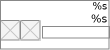
VISUALIZATION VIS_SENSOR_ROUND_RightAboveCheckQuerry  // 110x50
VAR_INPUT
    ITF_SENSOR_IN   :   ITF_SENSOR;
	stExklParameter	:	STRING [40];	
END_VAR
    Frame (0,0 110x50)
        shows VIS_SENSOR_ROUND_RightAboveCheckIsEnabled(ITF_SENSOR_IN := ITF_SENSOR_IN, stExklParameter := stExklParameter)
END_VISUALIZATION

// 40 Visualizations/ICON/SENSOR_FLAT/SENSOR_FLAT_TXT_RIGHT/BELOW/VIS_SENSOR_FLAT_RIGHT_BELOW
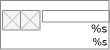
VISUALIZATION VIS_SENSOR_FLAT_RIGHT_BELOW  // 110x50
VAR_INPUT
    ITF_SENSOR_IN   :   ITF_SENSOR;	
END_VAR
VAR_INPUT CONSTANT	
	stExklParameter	:	STRING [40] := ' ';	
END_VAR
VAR CONSTANT
	uiIconNr		:	UINT := 3;
END_VAR
    Frame (0,0 110x50), invisible if: NOT fcCheckQuerryAndIconReturn(_ITF_IN := ITF_SENSOR_IN, _uiIconNr_IN := uiIconNr)
        shows VIS_SENSOR_FLAT_RigthBelowCheckQuerry(ITF_SENSOR_IN := ITF_SENSOR_IN, stExklParameter := stExklParameter)
END_VISUALIZATION

// 40 Visualizations/ICON/SENSOR_FLAT/SENSOR_FLAT_TXT_RIGHT/BELOW/VIS_SENSOR_FLAT_RigthBelowCheckIsEnabled
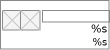
VISUALIZATION VIS_SENSOR_FLAT_RigthBelowCheckIsEnabled  // 110x50
VAR_INPUT
    ITF_SENSOR_IN   :   ITF_SENSOR;
	stExklParameter	:	STRING [40];	
END_VAR
    Frame (2,10 38x20), invisible if: NOT ITF_SENSOR_IN.proIsEnabled
        shows SensorFlat(ITF_SENSORIN := ITF_SENSOR_IN)
    Frame (42,10 68x40), invisible if: NOT ITF_SENSOR_IN.proIsEnabled
        shows ValueDwnUp(ITF_SENSORIN := ITF_SENSOR_IN, uiTextAusrichtung := 4)
    Rectangle (0,0 110x50)
        OnMouseClick:  Dialog=POPUP_SENSOR, Parameters={stExklParameter: stExklParameter, ITF_SENSORIN: ITF_SENSOR_IN, uiPopUpGruppe: 0}, OpenCentered=True
END_VISUALIZATION

// 40 Visualizations/ICON/SENSOR_FLAT/SENSOR_FLAT_TXT_RIGHT/BELOW/VIS_SENSOR_FLAT_RigthBelowCheckQuerry
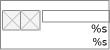
VISUALIZATION VIS_SENSOR_FLAT_RigthBelowCheckQuerry  // 110x50
VAR_INPUT
    ITF_SENSOR_IN   :   ITF_SENSOR;	
	stExklParameter	:	STRING [40];	
END_VAR
    Frame (0,0 110x50)
        shows VIS_SENSOR_FLAT_RigthBelowCheckIsEnabled(ITF_SENSOR_IN := ITF_SENSOR_IN, stExklParameter := stExklParameter)
END_VISUALIZATION

// 40 Visualizations/ICON/SENSOR_ROUND/SENSOR_ROUND_TXT_RIGHT/BELOW/VIS_SENSOR_ROUND_RIGHT_BELOW
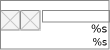
VISUALIZATION VIS_SENSOR_ROUND_RIGHT_BELOW  // 110x50
VAR_INPUT
    ITF_SENSOR_IN   :   ITF_SENSOR;	
END_VAR
VAR_INPUT CONSTANT	
	stExklParameter	:	STRING [40] := ' ';	
END_VAR
VAR CONSTANT
	uiIconNr		:	UINT := 5;
END_VAR
    Frame (0,0 110x50), invisible if: NOT fcCheckQuerryAndIconReturn(_ITF_IN := ITF_SENSOR_IN, _uiIconNr_IN := uiIconNr)
        shows VIS_SENSOR_ROUND_RightBelowCheckQuerry(ITF_SENSOR_IN := ITF_SENSOR_IN, stExklParameter := stExklParameter)
END_VISUALIZATION

// 40 Visualizations/ICON/SENSOR_BASE/ICON/Value/ValueDwnUp
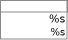
VISUALIZATION ValueDwnUp  // 68x40
VAR_INPUT
    ITF_SENSORIN   :   ITF_SENSOR;	
END_VAR
VAR_INPUT CONSTANT
    uiTextAusrichtung   : UINT := 4;    // 0 = Oben links | 1 = Horizontal zentriert | 2 = Rechts | 4 = Vertikal zentriert | 8 = Unten
END_VAR
    Frame (0,0 68x12)
        shows CtaSysSensorReCalculation.ValueRC(ITF_SENSOR_RE_CALCULATE := ITF_SENSORIN.ITF_RC, uiTextAusrichtung := uiTextAusrichtung)
    Textfield (0,13 68x12), "%s", text variable: ITF_SENSORIN.proSoftwareValue
        p3718999670: uiTextAusrichtung
    Textfield (0,26 68x12), "%s", text variable: ITF_SENSORIN.proGetBMK, invisible if: ITF_SENSORIN.proNoBmkInList
        p3718999670: uiTextAusrichtung
END_VISUALIZATION

// 40 Visualizations/ICON/SENSOR_BASE/ICON/Round/SensorRound
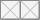
VISUALIZATION SensorRound  // 40x20
VAR_INPUT
    ITF_SENSORIN   :   ITF_SENSOR;	
END_VAR
    Ellipse (10,0 20x20), colour toggle: ITF_SENSORIN.proAcknowlege, invisible if: ITF_SENSORIN.proIsError
    Ellipse (10,0 20x20), colour toggle: ITF_SENSORIN.proIsError
    Image (0,0 20x20), invisible if: NOT ITF_SENSORIN.proIsWarning, image: CtaVisSymbols.ImagePool.CtaWarning
    Image (20,0 20x20), invisible if: NOT ITF_SENSORIN.proIsHandOnOrOff, image: CtaVisSymbols.ImagePool.front_hand_Yellow
    Image (20,0 20x20), invisible if: NOT ITF_SENSORIN.proHandOff, image: CtaVisSymbols.ImagePool.front_hand_Yellow_Off
END_VISUALIZATION

// 40 Visualizations/ICON/SENSOR_ROUND/SENSOR_ROUND_TXT_RIGHT/BELOW/VIS_SENSOR_ROUND_RightBelowCheckQuerry
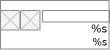
VISUALIZATION VIS_SENSOR_ROUND_RightBelowCheckQuerry  // 110x50
VAR_INPUT
    ITF_SENSOR_IN   :   ITF_SENSOR;
	stExklParameter	:	STRING [40];	
END_VAR
    Frame (0,0 110x50)
        shows VIS_SENSOR_ROUND_RightBelowCheckIsEnabled(ITF_SENSOR_IN := ITF_SENSOR_IN, stExklParameter := stExklParameter)
END_VISUALIZATION

// 40 Visualizations/ICON/SENSOR_ROUND/SENSOR_ROUND_TXT_RIGHT/BELOW/VIS_SENSOR_ROUND_RightBelowCheckIsEnabled
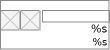
VISUALIZATION VIS_SENSOR_ROUND_RightBelowCheckIsEnabled  // 110x50
VAR_INPUT
    ITF_SENSOR_IN   :   ITF_SENSOR;
	stExklParameter	:	STRING [40];	
END_VAR
    Frame (0,10 40x20), invisible if: NOT ITF_SENSOR_IN.proIsEnabled
        shows SensorRound(ITF_SENSORIN := ITF_SENSOR_IN)
    Frame (42,10 68x40), invisible if: NOT ITF_SENSOR_IN.proIsEnabled
        shows ValueDwnUp(ITF_SENSORIN := ITF_SENSOR_IN, uiTextAusrichtung := 4)
    Rectangle (0,0 110x50)
        OnMouseClick:  Dialog=POPUP_SENSOR, Parameters={stExklParameter: , ITF_SENSORIN: ITF_SENSOR_IN, uiPopUpGruppe: 0}, OpenCentered=True
END_VISUALIZATION

// 40 Visualizations/ICON/SENSOR_ROUND/SENSOR_ROUNF_TXT_LEFT/BELOW/VIS_SENSOR_ROUND_LEFT_BELOW
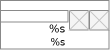
VISUALIZATION VIS_SENSOR_ROUND_LEFT_BELOW  // 110x50
VAR_INPUT
    ITF_SENSOR_IN   :   ITF_SENSOR;	
END_VAR
VAR_INPUT CONSTANT	
	stExklParameter	:	STRING [40] := ' ';	
END_VAR
VAR CONSTANT
	uiIconnr		:	UINT := 7;
END_VAR
    Frame (0,0 110x50), invisible if: NOT fcCheckQuerryAndIconReturn(_ITF_IN := ITF_SENSOR_IN, _uiIconNr_IN := uiIconNr)
        shows VIS_SENSOR_ROUND_LeftBelowCheckQuerry(ITF_SENSOR_IN := ITF_SENSOR_IN, stExklParameter := stExklParameter)
END_VISUALIZATION

// 40 Visualizations/ICON/SENSOR_ROUND/SENSOR_ROUNF_TXT_LEFT/BELOW/VIS_SENSOR_ROUND_LeftBelowCheckIsEnabled
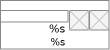
VISUALIZATION VIS_SENSOR_ROUND_LeftBelowCheckIsEnabled  // 110x50
VAR_INPUT
    ITF_SENSOR_IN   :   ITF_SENSOR;
	stExklParameter	:	STRING [40];	
END_VAR
    Frame (69,10 40x20), invisible if: NOT ITF_SENSOR_IN.proIsEnabled
        shows SensorRound(ITF_SENSORIN := ITF_SENSOR_IN)
    Frame (0,10 68x40), invisible if: NOT ITF_SENSOR_IN.proIsEnabled
        shows ValueDwnUp(ITF_SENSORIN := ITF_SENSOR_IN, uiTextAusrichtung := 6)
    Rectangle (0,0 110x50)
        OnMouseClick:  Dialog=POPUP_SENSOR, Parameters={stExklParameter: stExklParameter, ITF_SENSORIN: ITF_SENSOR_IN, uiPopUpGruppe: 0}, OpenCentered=True
END_VISUALIZATION

// 40 Visualizations/ICON/SENSOR_ROUND/SENSOR_ROUNF_TXT_LEFT/BELOW/VIS_SENSOR_ROUND_LeftBelowCheckQuerry
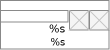
VISUALIZATION VIS_SENSOR_ROUND_LeftBelowCheckQuerry  // 110x50
VAR_INPUT
    ITF_SENSOR_IN   :   ITF_SENSOR;
	stExklParameter	:	STRING [40];	
END_VAR
    Frame (0,0 110x50)
        shows VIS_SENSOR_ROUND_LeftBelowCheckIsEnabled(ITF_SENSOR_IN := ITF_SENSOR_IN, stExklParameter := stExklParameter)
END_VISUALIZATION

// 40 Visualizations/POPUP/PARAMETER/IO_Parameter/VIS_SENSOR_IO_PARAMETER
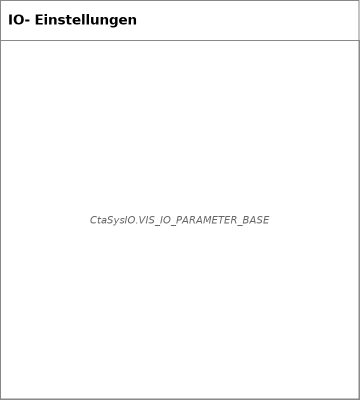
VISUALIZATION VIS_SENSOR_IO_PARAMETER  // 360x400
VAR_INPUT
    ITF_SENSORIN 	: 	ITF_SENSOR;
END_VAR
    Frame (0,40 360x360)
        shows CtaSysIO.VIS_IO_PARAMETER_BASE(ITF_IO_IN := ITF_SENSORIN.proSensorITF)
        shows AT_ParameterIO1(ITF_Parameter := ITF_Parameter)
    Label (5,0 150x40), "IO- Einstellungen"
END_VISUALIZATION

// 40 Visualizations/POPUP/OVERVIEW/VIS_SENSOR_OVERVIEW0
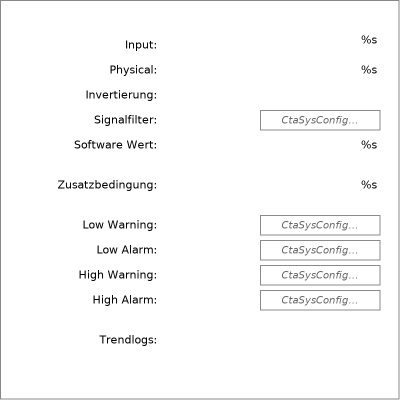
VISUALIZATION VIS_SENSOR_OVERVIEW0  // 400x400
VAR_INPUT
    ITF_SENSORIN	:	ITF_SENSOR;
END_VAR
    Textfield (5,0 385x30), text list: 'ValueInputType', text index: ITF_SENSORIN.proValueInputType
    Label (0,35 160x20), "Input:"
    Textfield (260,30 120x20), "%s", text variable: ITF_SENSORIN.proPhysicalValue
    Label (0,60 160x20), "Physical:"
    Textfield (260,60 120x20), "%s", text variable: ITF_SENSORIN.proRawValue
    Label (0,85 160x20), "Invertierung:", invisible if: ITF_SENSORIN.proValueInputType <> 4
    Textfield (165,85 60x20), invisible if: ITF_SENSORIN.proValueInputType <> 4, text list: 'WarnungsStatus', text index: ITF_SENSORIN.proInvertierung
    Label (0,110 160x20), "Signalfilter:", invisible if: (ITF_SENSORIN.proValueInputType = 2) OR (ITF_SENSORIN.proValueInputType = 4)
    Textfield (165,110 60x20), invisible if: (ITF_SENSORIN.proValueInputType = 2) OR (ITF_SENSORIN.proValueInputType = 4), text list: 'WarnungsStatus', text index: CtaSysConfig.fcGetEnumerationId(ITF_SENSORIN.P_scFilter_fbxEnabled)
    Frame (260,110 120x20), invisible if: ITF_SENSORIN.proValueInputType = 2 OR ITF_SENSORIN.proValueInputType = 4 OR (CtaSysConfig.fcGetEnumerationId(ITF_SENSORIN.P_scFilter_fbxEnabled) <>1)
        shows CtaSysConfig.visSHOWDATA(visfbDATATYPEIn := ITF_SENSORIN.P_scFilter_fbrValue)
    Label (0,135 160x20), "Software Wert:"
    Textfield (260,135 120x20), "%s", text variable: ITF_SENSORIN.proSoftwareValue, input disabled if: TRUE
    Label (0,175 160x20), "Zusatzbedingung:"
    Textfield (165,175 60x20), text list: 'WarnungsStatus', text index: CtaSysConfig.fcGetEnumerationId(ITF_SENSORIN.P_scAlCondition_fbxEnable)
    Label (0,215 160x20), "Low Warning:"
    Textfield (165,215 60x20), text list: 'WarnungsStatus', text index: CtaSysConfig.fcGetEnumerationId(ITF_SENSORIN.P_scLoWarning_fbxDoesWarning)
    Frame (260,215 120x20), invisible if: (CtaSysConfig.fcGetEnumerationId(ITF_SENSORIN.P_scLoWarning_fbxDoesWarning)<>1)
        shows CtaSysConfig.visSHOWDATA(visfbDATATYPEIn := ITF_SENSORIN.P_scLoWarning_fbrValue)
    Label (0,240 160x20), "Low Alarm:"
    Textfield (165,240 60x20), text list: 'WarnungsStatus', text index: CtaSysConfig.fcGetEnumerationId(ITF_SENSORIN.P_scLoAlarm_fbxDoesAlarm)
    Frame (260,240 120x20), invisible if: (CtaSysConfig.fcGetEnumerationId(ITF_SENSORIN.P_scLoAlarm_fbxDoesAlarm)<>1)
        shows CtaSysConfig.visSHOWDATA(visfbDATATYPEIn := ITF_SENSORIN.P_scLoAlarm_fbrValue)
    Label (0,265 160x20), "High Warning:"
    Textfield (165,265 60x20), text list: 'WarnungsStatus', text index: CtaSysConfig.fcGetEnumerationId(ITF_SENSORIN.P_scHighWarning_fbxDoesWarning)
    Frame (260,265 120x20), invisible if: (CtaSysConfig.fcGetEnumerationId(ITF_SENSORIN.P_scHighWarning_fbxDoesWarning)<>1)
        shows CtaSysConfig.visSHOWDATA(visfbDATATYPEIn := ITF_SENSORIN.P_scHighWarning_fbrValue)
    Label (0,290 160x20), "High Alarm:"
    Textfield (165,290 60x20), text list: 'WarnungsStatus', text index: CtaSysConfig.fcGetEnumerationId(ITF_SENSORIN.P_scHighAlram_fbxDoesAlarm)
    Frame (260,290 120x20), invisible if: (CtaSysConfig.fcGetEnumerationId(ITF_SENSORIN.P_scHighAlram_fbxDoesAlarm)<>1)
        shows CtaSysConfig.visSHOWDATA(visfbDATATYPEIn := ITF_SENSORIN.P_scHighAlarm_fbrValue)
    Label (0,330 160x20), "Trendlogs:"
    Textfield (165,330 60x20), text list: 'WarnungsStatus', text index: CtaSysConfig.fcGetEnumerationId(ITF_SENSORIN.P_scInfluxDb_fbxEnable)
    Textfield (260,175 120x20), "%s", text variable: BOOL_TO_STRING(ITF_SENSORIN.proxErrorConditionValue), invisible if: (CtaSysConfig.fcGetEnumerationId(ITF_SENSORIN.P_scAlCondition_fbxEnable)<>1), input disabled if: TRUE
END_VISUALIZATION

// 40 Visualizations/POPUP/BUS/Sensor_BUS_CS
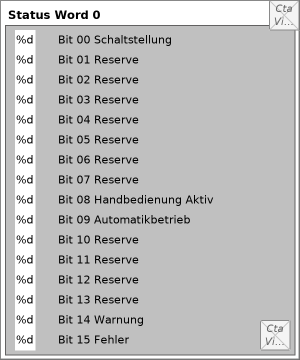
VISUALIZATION Sensor_BUS_CS  // 300x360
VAR_INPUT
    ITF_SENSORIN    :   ITF_SENSOR;
    ayControllWord  :   REFERENCE TO ARRAY[0..3] OF WORD;
    ayStateWord     :   REFERENCE TO ARRAY[0..3] OF WORD;
END_VAR
VAR
    xShowCw :   BOOL;
	xShowCw1:   BOOL;
	xShowCw2:   BOOL;
	xShowCw3:   BOOL;
    xShowSw :   BOOL;
    xShowSw1:   BOOL;
    xShowSw2:   BOOL;
	xShowSw3:   BOOL;
END_VAR
    Textfield (0,10 130x20), "%b", text variable: ayControllWord[0], invisible if: TRUE, input disabled if: TRUE
    Label (140,10 120x20), "Controll Word 0", invisible if: TRUE
    Image (266,5 30x30), invisible if: TRUE, input disabled if: TRUE, image: CtaVisSymbols.ImagePool.information-variant
        OnMouseClick: execute {
            xShowCw := TRUE;
            xShowCw1:= FALSE;
            xShowCw2:= FALSE;
            xShowCw3:= FALSE;
            xShowSw := FALSE;
            xShowSw1:= FALSE;
            xShowSw2:= FALSE;
            xShowSW3:= FALSE;
        }
    Textfield (0,50 130x20), "%d", text variable: ayControllWord[1], invisible if: TRUE, input disabled if: TRUE
    Label (140,50 120x20), "Controll Word 1", invisible if: TRUE
    Textfield (0,90 130x20), "%d", text variable: ayControllWord[2], invisible if: TRUE, input disabled if: TRUE
    Label (140,90 120x20), "Controll Word 2", invisible if: TRUE
    Textfield (0,130 130x20), "%d", text variable: ayControllWord[3], invisible if: TRUE, input disabled if: TRUE
    Label (140,130 120x20), "Controll Word 3", invisible if: TRUE
    Textfield (0,170 130x20), "%b", text variable: ayStateWord[0]
        OnMouseDown: write the text variable via Default
    Label (140,170 120x20), "State Word 0"
    Image (265,165 30x30), image: CtaVisSymbols.ImagePool.information-variant
        OnMouseClick: execute {
            xShowCw := FALSE;
            xShowCw1:= FALSE;
            xShowCw2:= FALSE;
            xShowCw3:= FALSE;
            xShowSw := TRUE;
            xShowSw1:= FALSE;
            xShowSw2:= FALSE;
            xShowSW3:= FALSE;
        }
    Textfield (0,210 130x20), "%d", text variable: ayStateWord[1]
    Label (140,210 120x20), "State Word 1"
    Image (265,205 30x30), image: CtaVisSymbols.ImagePool.information-variant
        OnMouseClick: execute {
            xShowCw := FALSE;
            xShowCw1:= FALSE;
            xShowCw2:= FALSE;
            xShowCw3:= FALSE;
            xShowSw := FALSE;
            xShowSw1:= TRUE;
            xShowSw2:= FALSE;
            xShowSW3:= FALSE;
        }
    Textfield (0,250 130x20), "%d", text variable: ayStateWord[2], invisible if: ITF_SENSORIN.proValueInputType = enInputType.DigitalInput OR ITF_SENSORIN.proValueInputType = enInputType.Digital_ITF_Input, input disabled if: ITF_SENSORIN.proValueInputType = enInputType.DigitalInput OR ITF_SENSORIN.proValueInputType = enInputType.Digital_ITF_Input
    Label (140,250 120x20), "State Word 2", invisible if: ITF_SENSORIN.proValueInputType = enInputType.DigitalInput OR ITF_SENSORIN.proValueInputType = enInputType.Digital_ITF_Input
    Image (265,245 30x30), invisible if: ITF_SENSORIN.proValueInputType = enInputType.DigitalInput OR ITF_SENSORIN.proValueInputType = enInputType.Digital_ITF_Input, input disabled if: ITF_SENSORIN.proValueInputType = enInputType.DigitalInput OR ITF_SENSORIN.proValueInputType = enInputType.Digital_ITF_Input, image: CtaVisSymbols.ImagePool.information-variant
        OnMouseClick: execute {
            xShowCw := FALSE;
            xShowCw1:= FALSE;
            xShowCw2:= FALSE;
            xShowCw3:= FALSE;
            xShowSw := FALSE;
            xShowSw1:= FALSE;
            xShowSw2:= TRUE;
            xShowSW3:= FALSE;
        }
    Textfield (0,290 130x20), "%d", text variable: ayStateWord[3]
    Label (140,289 120x20), "State Word 3"
    Image (265,285 30x30), image: CtaVisSymbols.ImagePool.information-variant
        OnMouseClick: execute {
            xShowCw := FALSE;
            xShowCw1:= FALSE;
            xShowCw2:= FALSE;
            xShowCw3:= FALSE;
            xShowSw := FALSE;
            xShowSw1:= FALSE;
            xShowSw2:= FALSE;
            xShowSW3:= TRUE;
        }
    Image (265,45 30x30), invisible if: TRUE, input disabled if: TRUE, image: CtaVisSymbols.ImagePool.information-variant
        OnMouseClick: execute {
            xShowCw := FALSE;
            xShowCw1:= TRUE;
            xShowCw2:= FALSE;
            xShowCw3:= FALSE;
            xShowSw := FALSE;
            xShowSw1:= FALSE;
            xShowSw2:= FALSE;
            xShowSW3:= FALSE;
        }
    Image (265,85 30x30), invisible if: TRUE, input disabled if: TRUE, image: CtaVisSymbols.ImagePool.information-variant
        OnMouseClick: execute {
            xShowCw := FALSE;
            xShowCw1:= FALSE;
            xShowCw2:= TRUE;
            xShowCw3:= FALSE;
            xShowSw := FALSE;
            xShowSw1:= FALSE;
            xShowSw2:= FALSE;
            xShowSW3:= FALSE;
        }
    Image (265,125 30x30), invisible if: TRUE, input disabled if: TRUE, image: CtaVisSymbols.ImagePool.information-variant
        OnMouseClick: execute {
            xShowCw := FALSE;
            xShowCw1:= FALSE;
            xShowCw2:= FALSE;
            xShowCw3:= TRUE;
            xShowSw := FALSE;
            xShowSw1:= FALSE;
            xShowSw2:= FALSE;
            xShowSW3:= FALSE;
        }
    Frame (0,0 300x360), invisible if: NOT xShowSw3
        shows Sensor_BUS_SW3_Detail(wDetail := ayStateWord[3], ITF_SENSORIN := ITF_SENSORIN, xShow := xShowSw3)
    Frame (0,0 300x360), invisible if: NOT xShowSw2
        shows Sensor_BUS_SW2_Detail(wDetail := ayStateWord[2], ITF_SENSORIN := ITF_SENSORIN, xShow := xShowSw2)
    Frame (0,0 300x360), invisible if: NOT xShowSw1
        shows Sensor_BUS_SW1_Detail(wDetail := ayStateWord[1], ITF_SENSORIN := ITF_SENSORIN, xShow := xShowSw1)
    Frame (0,0 300x360), invisible if: NOT xShowSw
        shows Sensor_BUS_SW0_Detail(wDetail := ayStateWord[0], ITF_SENSORIN := ITF_SENSORIN, xShow := xShowSw)
END_VISUALIZATION

// 40 Visualizations/POPUP/BUS/Sensor_BUS
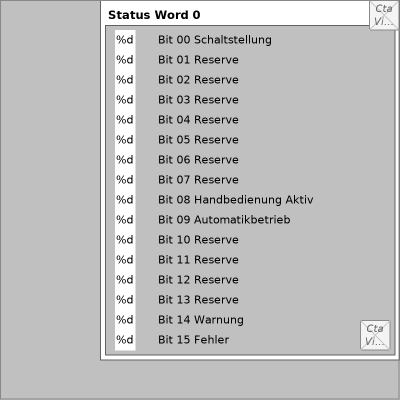
VISUALIZATION Sensor_BUS  // 400x400
VAR_INPUT
    ITF_SENSORIN    :   ITF_SENSOR;	
END_VAR
    Frame (100,0 300x360)
        shows Sensor_BUS_CS(ITF_SENSORIN := ITF_SENSORIN, ayControllWord := ITF_SENSORIN.proModbusControllWord, ayStateWord := ITF_SENSORIN.proModbusStateWord)
END_VISUALIZATION

// 40 Visualizations/POPUP/BUS/Sensor_BUS_SW0_Detail
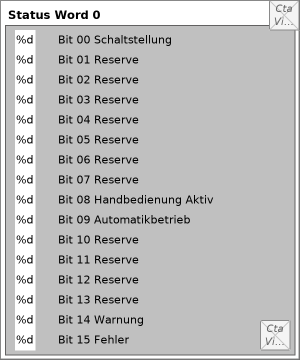
VISUALIZATION Sensor_BUS_SW0_Detail  // 300x360
VAR_IN_OUT
    wDetail     :   WORD;
END_VAR
VAR_INPUT	
    ITF_SENSORIN    :   ITF_SENSOR;
END_VAR
VAR_IN_OUT
    xShow       :   BOOL;
END_VAR
    RoundedRectangle (0,0 300x360)
    RoundedRectangle (5,25 290x330)
    Textfield (15,30 20x20), "%d", text variable: TO_WORD(wDetail.0), input disabled if: NOT ITF_SENSORIN.proModbusTest
        OnMouseClick: execute { wDetail.0 := NOT wDetail.0; }
    Label (55,30 220x20), "Bit 00 Schaltstellung"
    Textfield (15,50 20x20), "%d", text variable: TO_WORD(wDetail.1), input disabled if: NOT ITF_SENSORIN.proModbusTest
        OnMouseClick: execute { wDetail.1 := NOT wDetail.1; }
    Label (55,50 220x20), "Bit 01 Reserve"
    Textfield (15,70 20x20), "%d", text variable: TO_WORD(wDetail.2), input disabled if: NOT ITF_SENSORIN.proModbusTest
        OnMouseClick: execute { wDetail.2 := NOT wDetail.2; }
    Label (55,70 220x20), "Bit 02 Reserve"
    Textfield (15,90 20x20), "%d", text variable: TO_WORD(wDetail.3), input disabled if: NOT ITF_SENSORIN.proModbusTest
        OnMouseClick: execute { wDetail.3 := NOT wDetail.3; }
    Label (55,90 220x20), "Bit 03 Reserve"
    Textfield (15,110 20x20), "%d", text variable: TO_WORD(wDetail.4), input disabled if: NOT ITF_SENSORIN.proModbusTest
        OnMouseClick: execute { wDetail.4 := NOT wDetail.4; }
    Label (55,110 220x20), "Bit 04 Reserve"
    Textfield (15,130 20x20), "%d", text variable: TO_WORD(wDetail.5), input disabled if: NOT ITF_SENSORIN.proModbusTest
        OnMouseClick: execute { wDetail.5 := NOT wDetail.5; }
    Label (55,130 220x20), "Bit 05 Reserve"
    Textfield (15,150 20x20), "%d", text variable: TO_WORD(wDetail.6), input disabled if: NOT ITF_SENSORIN.proModbusTest
        OnMouseClick: execute { wDetail.6 := NOT wDetail.6; }
    Label (55,150 220x20), "Bit 06 Reserve"
    Textfield (15,170 20x20), "%d", text variable: TO_WORD(wDetail.7), input disabled if: NOT ITF_SENSORIN.proModbusTest
        OnMouseClick: execute { wDetail.7 := NOT wDetail.7; }
    Label (55,170 220x20), "Bit 07 Reserve"
    Textfield (15,190 20x20), "%d", text variable: TO_WORD(wDetail.8), input disabled if: NOT ITF_SENSORIN.proModbusTest
        OnMouseClick: execute { wDetail.8 := NOT wDetail.8; }
    Label (55,190 220x20), "Bit 08 Handbedienung Aktiv"
    Textfield (15,210 20x20), "%d", text variable: TO_WORD(wDetail.9), input disabled if: NOT ITF_SENSORIN.proModbusTest
        OnMouseClick: execute { wDetail.9 := NOT wDetail.9; }
    Label (55,210 220x20), "Bit 09 Automatikbetrieb"
    Textfield (15,230 20x20), "%d", text variable: TO_WORD(wDetail.10), input disabled if: NOT ITF_SENSORIN.proModbusTest
        OnMouseClick: execute { wDetail.10 := NOT wDetail.10; }
    Label (55,230 220x20), "Bit 10 Reserve"
    Textfield (15,250 20x20), "%d", text variable: TO_WORD(wDetail.11), input disabled if: NOT ITF_SENSORIN.proModbusTest
        OnMouseClick: execute { wDetail.11 := NOT wDetail.11; }
    Label (55,250 220x20), "Bit 11 Reserve"
    Textfield (15,270 20x20), "%d", text variable: TO_WORD(wDetail.12), input disabled if: NOT ITF_SENSORIN.proModbusTest
        OnMouseClick: execute { wDetail.12 := NOT wDetail.12; }
    Label (55,270 220x20), "Bit 12 Reserve"
    Textfield (15,290 20x20), "%d", text variable: TO_WORD(wDetail.13), input disabled if: NOT ITF_SENSORIN.proModbusTest
        OnMouseClick: execute { wDetail.13 := NOT wDetail.13; }
    Label (55,290 220x20), "Bit 13 Reserve"
    Textfield (15,310 20x20), "%d", text variable: TO_WORD(wDetail.14), input disabled if: NOT ITF_SENSORIN.proModbusTest
        OnMouseClick: execute { wDetail.14 := NOT wDetail.14; }
    Label (55,310 220x20), "Bit 14 Warnung"
    Textfield (15,330 20x20), "%d", text variable: TO_WORD(wDetail.15), input disabled if: NOT ITF_SENSORIN.proModbusTest
        OnMouseClick: execute { wDetail.15 := NOT wDetail.15; }
    Label (55,330 220x20), "Bit 15 Fehler"
    Image (269,0 30x30), image: CtaVisSymbols.ImagePool.close_solo_black
        OnMouseClick: execute { xShow := FALSE; ITF_SENSORIN.proModbusTest := FALSE; }
    Label (5,0 150x30), "Status Word 0"
    Image (260,320 30x30), invisible if: ITF_SENSORIN.proModbusTest, image: CtaVisSymbols.ImagePool.front_hand_Black
        OnMouseClick: execute { ITF_SENSORIN.proModbusTest := TRUE; }
    Image (260,320 30x30), invisible if: NOT ITF_SENSORIN.proModbusTest, image: CtaVisSymbols.ImagePool.front_hand_Yellow
        OnMouseClick: execute { ITF_SENSORIN.proModbusTest := False; }
END_VISUALIZATION

// 40 Visualizations/POPUP/BUS/Sensor_BUS_SW1_Detail
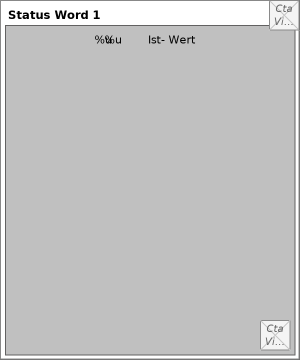
VISUALIZATION Sensor_BUS_SW1_Detail  // 300x360
VAR_IN_OUT
    wDetail     :   WORD;
END_VAR
VAR_INPUT	
    ITF_SENSORIN    :   ITF_SENSOR;
END_VAR
VAR_IN_OUT
    xShow       :   BOOL;
END_VAR
    RoundedRectangle (0,0 300x360)
    RoundedRectangle (5,25 290x330)
    Image (269,0 30x30), image: CtaVisSymbols.ImagePool.close_solo_black
        OnMouseClick: execute { xShow := FALSE; ITF_SENSORIN.proModbusTest := FALSE; }
    Label (5,0 150x30), "Status Word 1"
    Label (145,30 120x20), "Ist- Wert"
    Textfield (5,30 110x20), "%u", text variable: wDetail, input disabled if: NOT ITF_SENSORIN.proModbusTest
        OnMouseClick: write the text variable via InputWithLimits, min 0, max 100
    Textfield (15,30 110x20), "%u", text variable: wDetail, invisible if: ITF_SENSORIN.proModbusTest
    Image (260,320 30x30), invisible if: ITF_SENSORIN.proModbusTest, image: CtaVisSymbols.ImagePool.front_hand_Black
        OnMouseClick: execute { ITF_SENSORIN.proModbusTest := TRUE; }
    Image (260,320 30x30), invisible if: NOT ITF_SENSORIN.proModbusTest, image: CtaVisSymbols.ImagePool.front_hand_Yellow
        OnMouseClick: execute { ITF_SENSORIN.proModbusTest := False; }
END_VISUALIZATION

// 40 Visualizations/POPUP/BUS/Sensor_BUS_SW2_Detail
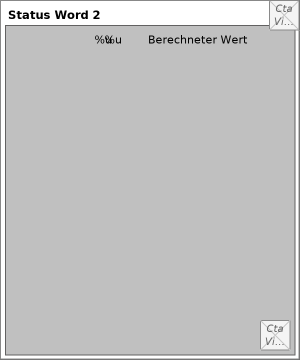
VISUALIZATION Sensor_BUS_SW2_Detail  // 300x360
VAR_IN_OUT
    wDetail             :   WORD;
END_VAR
VAR_INPUT	
    ITF_SENSORIN       :   ITF_SENSOR;
END_VAR
VAR_IN_OUT
    xShow               :   BOOL;
END_VAR
    RoundedRectangle (0,0 300x360)
    RoundedRectangle (5,25 290x330)
    Image (269,0 30x30), image: CtaVisSymbols.ImagePool.close_solo_black
        OnMouseClick: execute { xShow := FALSE; ITF_SENSORIN.proModbusTest := FALSE; }
    Label (5,0 150x30), "Status Word 2"
    Label (145,30 120x20), "Berechneter Wert"
    Textfield (5,30 110x20), "%u", text variable: wDetail, input disabled if: NOT ITF_SENSORIN.proModbusTest
        OnMouseClick: write the text variable via InputWithLimits, min 0, max 100
    Textfield (15,30 110x20), "%u", text variable: wDetail, invisible if: ITF_SENSORIN.proModbusTest
    Image (260,320 30x30), invisible if: ITF_SENSORIN.proModbusTest, image: CtaVisSymbols.ImagePool.front_hand_Black
        OnMouseClick: execute { ITF_SENSORIN.proModbusTest := TRUE; }
    Image (260,320 30x30), invisible if: NOT ITF_SENSORIN.proModbusTest, image: CtaVisSymbols.ImagePool.front_hand_Yellow
        OnMouseClick: execute { ITF_SENSORIN.proModbusTest := False; }
END_VISUALIZATION

// 40 Visualizations/POPUP/BUS/Sensor_BUS_SW3_Detail
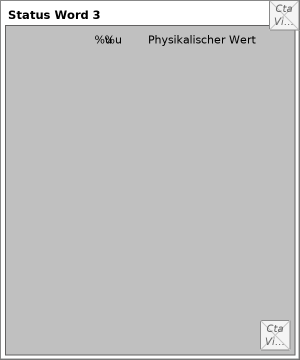
VISUALIZATION Sensor_BUS_SW3_Detail  // 300x360
VAR_IN_OUT
    wDetail             :   WORD;
END_VAR
VAR_INPUT	
    ITF_SENSORIN       :   ITF_SENSOR;
END_VAR
VAR_IN_OUT
    xShow               :   BOOL;
END_VAR
    RoundedRectangle (0,0 300x360)
    RoundedRectangle (5,25 290x330)
    Image (269,0 30x30), image: CtaVisSymbols.ImagePool.close_solo_black
        OnMouseClick: execute { xShow := FALSE; ITF_SENSORIN.proModbusTest := FALSE; }
    Label (5,0 150x30), "Status Word 3"
    Label (145,30 120x20), "Physikalischer Wert"
    Textfield (5,30 110x20), "%u", text variable: wDetail, input disabled if: NOT ITF_SENSORIN.proModbusTest
        OnMouseClick: write the text variable via InputWithLimits, min 0, max 100
    Textfield (15,30 110x20), "%u", text variable: wDetail, invisible if: ITF_SENSORIN.proModbusTest
    Image (260,320 30x30), invisible if: ITF_SENSORIN.proModbusTest, image: CtaVisSymbols.ImagePool.front_hand_Black
        OnMouseClick: execute { ITF_SENSORIN.proModbusTest := TRUE; }
    Image (260,320 30x30), invisible if: NOT ITF_SENSORIN.proModbusTest, image: CtaVisSymbols.ImagePool.front_hand_Yellow
        OnMouseClick: execute { ITF_SENSORIN.proModbusTest := False; }
END_VISUALIZATION

// 40 Visualizations/ICON/SENSOR_BASE/ICON/Value/ValueUpDwn
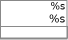
VISUALIZATION ValueUpDwn  // 68x40
VAR_INPUT
    ITF_SENSORIN   :   ITF_SENSOR;	
END_VAR
VAR_INPUT CONSTANT
    uiTextAusrichtung   : UINT := 4;    // 0 = Oben links | 1 = Horizontal zentriert | 2 = Rechts | 4 = Vertikal zentriert | 8 = Unten
END_VAR
    Textfield (0,0 68x12), "%s", text variable: ITF_SENSORIN.proGetBMK, invisible if: ITF_SENSORIN.proNoBmkInList
        p3718999670: uiTextAusrichtung
    Textfield (0,13 68x12), "%s", text variable: ITF_SENSORIN.proSoftwareValue
        p3718999670: uiTextAusrichtung
    Frame (0,26 68x12)
        shows CtaSysSensorReCalculation.ValueRC(ITF_SENSOR_RE_CALCULATE := ITF_SENSORIN.ITF_RC, uiTextAusrichtung := uiTextAusrichtung)
END_VISUALIZATION

// 40 Visualizations/ICON/SENSOR_FLAT/SENSOR_FLAT_TXT_LEFT/MIDDLE/VIS_SENSOR_FLAT_LeftMiddleCheckIsEnabled
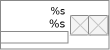
VISUALIZATION VIS_SENSOR_FLAT_LeftMiddleCheckIsEnabled  // 110x50
VAR_INPUT
    ITF_SENSOR_IN   :   ITF_SENSOR;
	stExklParameter	:	STRING [40];	
END_VAR
    Frame (70,15 38x20), invisible if: NOT ITF_SENSOR_IN.proIsEnabled
        shows SensorFlat(ITF_SENSORIN := ITF_SENSOR_IN)
    Frame (0,5 68x40), invisible if: NOT ITF_SENSOR_IN.proIsEnabled
        shows ValueUpDwn(ITF_SENSORIN := ITF_SENSOR_IN, uiTextAusrichtung := 6)
    Rectangle (0,0 110x50)
        OnMouseClick:  Dialog=POPUP_SENSOR, Parameters={stExklParameter: stExklParameter, ITF_SENSORIN: ITF_SENSOR_IN, uiPopUpGruppe: 0}, OpenCentered=True
END_VISUALIZATION

// 40 Visualizations/ICON/SENSOR_FLAT/SENSOR_FLAT_TXT_LEFT/MIDDLE/VIS_SENSOR_FLAT_LeftMiddleCheckQuerry
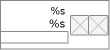
VISUALIZATION VIS_SENSOR_FLAT_LeftMiddleCheckQuerry  // 110x50
VAR_INPUT
    ITF_SENSOR_IN   :   ITF_SENSOR;
	stExklParameter	:	STRING [40];	
END_VAR
    Frame (0,0 110x50)
        shows VIS_SENSOR_FLAT_LeftMiddleCheckIsEnabled(ITF_SENSOR_IN := ITF_SENSOR_IN, stExklParameter := stExklParameter)
END_VISUALIZATION

// 40 Visualizations/ICON/SENSOR_FLAT/SENSOR_FLAT_TXT_LEFT/MIDDLE/VIS_SENSOR_FLAT_LEFT_MIDDLE
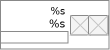
VISUALIZATION VIS_SENSOR_FLAT_LEFT_MIDDLE  // 110x50
VAR_INPUT
    ITF_SENSOR_IN   :   ITF_SENSOR;	
END_VAR
VAR_INPUT CONSTANT	
	stExklParameter	:	STRING [40] := ' ';	
END_VAR
VAR CONSTANT
	uiIconNr		: UINT := 0;
END_VAR
    Frame (0,0 110x50), invisible if: NOT fcCheckQuerryAndIconReturn(_ITF_IN := ITF_SENSOR_IN, _uiIconNr_IN := uiIconNr)
        shows VIS_SENSOR_FLAT_LeftMiddleCheckQuerry(ITF_SENSOR_IN := ITF_SENSOR_IN, stExklParameter := stExklParameter)
END_VISUALIZATION

// 40 Visualizations/ICON/SENSOR_FLAT/SENSOR_FLAT_TXT_RIGHT/MIDDLE/VIS_SENSOR_FLAT_RIGHT_MIDDLE
